{attribute 'linkalways'}
{attribute 'hide_all_locals'}
FUNCTION_BLOCK ABSTRACT ValueBase IMPLEMENTS ValueWithType
VAR
	_ValueType : ValueType;
END_VAR

{attribute 'monitoring' := 'call'}
PROPERTY ValueType : ValueType
GET
ValueType := _ValueType;
END_GET
END_PROPERTY

END_FUNCTION_BLOCK

(* stored: Version 1.1.0.1, ProductVersion 3.1.4024.15
   POU ValueBase: Id {6e437225-aae5-40c6-9153-868cb94efe47}, SpecialFunc None
   Property ValueType: Id {3135a025-3087-412d-807e-194fe88e262c}
   Get Get: Id {e4a8edd3-49e5-4d57-b9f9-fa09826b7b04} *)
